{attribute 'GeneratedUsingTerminal: AMI8000-0000-0016'}
{attribute addProperty BoxType "AMI8000-0000-0016"}
{attribute addProperty Id "ControlwordAT %Q*UINT2"}
{attribute addProperty CRC "4092675873"}
{attribute addProperty Size "2"}
TYPE DRV_Controlword_F3F14721 :
STRUCT
	{attribute addProperty Name "Controlword"}
	Controlword AT %Q* : UINT;
END_STRUCT
END_TYPE

(* stored: Version 1.2.0.0, ProductVersion 3.1.4024.9
   DUT DRV_Controlword_F3F14721: Id {2cdfe20c-0094-416a-ad17-ef7edf678acd} *)
